FUNCTION_BLOCK FB_Maschinentuer
VAR_INPUT
	//Steuereingänge //Außenbefehle
	bOpen :BOOL; 
	bClose :BOOL;
	bEnable :BOOL; // Zur Machinenfreigabe
	
	//Sensoreingänge
	bDoorC :BOOL;
	bDoorO :BOOL;
END_VAR
VAR_OUTPUT
	//Aktor Ausgang
	bVentil :BOOL;
	//Zustände
	bError :BOOL;
	
END_VAR
VAR
	nState :INT :=0;
END_VAR



CASE nState OF 
	0: // Tür geschlossen Zustand
	// Ausgänge setzen
	bVentil := TRUE;
	
	// Übergangsbedingung 
	IF NOT bDoorC AND bEnable THEN
		nState :=3; // Tür schließen
	ELSIF bOpen THEN
		nState:=1;	// Tür öffnen
	END_IF
	1:// Tür öffnen
	// Ausgänge setzen
	bVentil :=FALSE;
	
	// Übergangsbedinugnen
	IF bDoorO THEN
		nState := 2; // Tür geöffnet
	END_IF
	2: // Tür geöffnet
	// Ausgänge setzen
	bVentil :=FALSE;
	
	// Übergangsbedinungen
	IF bClose AND bEnable THEN
		nState :=3; // Tür schließen
	END_IF
	3:// Tür schließen
	// Ausgänge setzen 
	bVentil :=TRUE;
	
	//Übergangsbedingung
	IF bDoorC THEN
		nState :=0; //Tür geschlossen
	END_IF
	
END_CASE

END_FUNCTION_BLOCK

(* stored: Version 1.1.0.1, ProductVersion 3.1.4024.15
   POU FB_Maschinentuer: Id {ff2d8ac9-d1b9-4363-a416-cd40268ac519}, SpecialFunc None *)
